TYPE RecvBuffer : ARRAY[1..RoboConnectParams.receiveBufferSize] OF BYTE; END_TYPE

(* stored: Version 1.1.0.1
   DUT RecvBuffer: Id {8995419b-89be-4df0-9b2d-e271f0a62774} *)
